(* IEC 61131-3 sources: InfiniteStateMachine/extracted_st/infinitestatemachine/function_blocks/statemachine/depth, 1 file *)

(* ---- Depth.st ---- *)
(* --- Interface --- *)
METHOD Depth : INT
VAR_INPUT
END_VAR

(* --- Implementation --- *)
Depth := iDepth;
